RoboDK station: Main.rdk

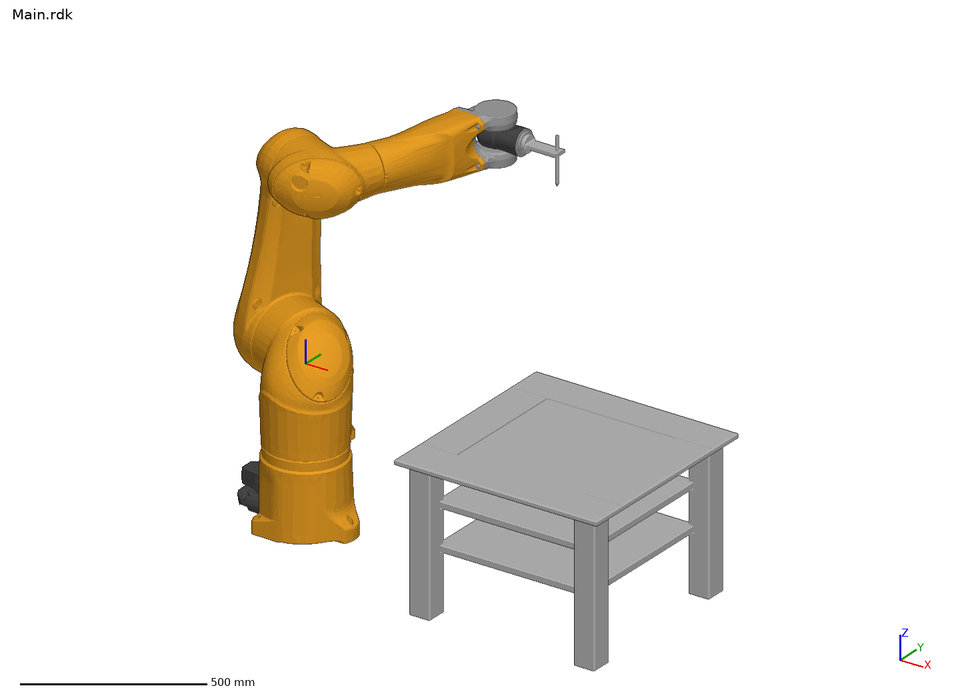
[picture v0: the station drawn from its stored meshes, robots at their saved joint values, targets as dots, program paths as lines]
Station Iteration1Übung0 (saved by RoboDK 5.6.9). Poses are relative to the parent item; angles as X-Y-Z fixed-axis rotations.
  - frame Staubli TX2-90L Base at (0, 0, 478) mm
    - robot Staubli TX2-90L: 6 axes, payload 5 kg, reach 1200 mm, repeatability 0.035 mm, weight 117 kg
        modified DH rows (alpha deg, a mm, theta deg, d mm): 0, 0, 0, 478; -90, 50, -90, 50; 0, 500, -90, 0; -90, 0, 0, 550; 90, 0, 0, 0; -90, 0, 180, 100
        base shift (0, 0, -478) mm
        joint limits [-180, -130, -145, -270, -115, -270] to [180, 147.5, 145, 270, 140, 270]; home [0, 0, 90, 0, 0, 0]; saved at [67.031, 3.495, 86.409, -89.959, 67.031, 89.895]
      - tool PenFixture, TCP at (100, 0, 100) mm, rotated rx 0 ry 90 rz 0 deg, size 150 x 50 x 110 mm, geometry from PenFixture.stl
  - object HolzTisch at (850, 0, 0) mm, size 660.1 x 660.1 x 466.4 mm, geometry from HolzTisch.stl
